// TIA Portal V20 export
DATA_BLOCK "DB_AsiSetpoint"   // DB32
// stored: Access Published, MemoryReserve 100, Namespace Global
   VAR
      Line : Struct
         A1 : Struct
            DirChange : Struct
               Conveyor : Array[_.gMinA1.._.gMaxA1] of Bool;
            END_STRUCT;
            Speed : Struct
               Conveyor : Array[_.gMinA1.._.gMaxA1] of Bool;
            END_STRUCT;
         END_STRUCT;
         B1 : Struct
            DirChange : Struct
               Conveyor : Array[_.gMinB1.._.gMaxB1] of Bool;
            END_STRUCT;
            Speed : Struct
               Conveyor : Array[_.gMinB1.._.gMaxB1] of Bool;
            END_STRUCT;
         END_STRUCT;
         C1 : Struct
            DirChange : Struct
               Conveyor : Array[_.gMinC1.._.gMaxC1] of Bool;
            END_STRUCT;
            Speed : Struct
               Conveyor : Array[_.gMinC1.._.gMaxC1] of Bool;
            END_STRUCT;
         END_STRUCT;
         D1 : Struct
            DirChange : Struct
               Conveyor : Array[_.gMinD1.._.gMaxD1] of Bool;
            END_STRUCT;
            Speed : Struct
               Conveyor : Array[_.gMinD1.._.gMaxD1] of Bool;
            END_STRUCT;
         END_STRUCT;
      END_STRUCT;
   END_VAR
BEGIN
   // Line.A1.DirChange.Conveyor[1001] : AS1.1.1
   // Line.A1.DirChange.Conveyor[1002] : AS1.1.2
   // Line.A1.Speed.Conveyor[1001] : AS1.1.1
   // Line.A1.Speed.Conveyor[1002] : AS1.1.2
END_DATA_BLOCK
